TYPE if_BitCommand_u :
UNION
    awPBOM : ARRAY[0..1] OF WORD;
    dwPBOM : DWORD;
END_UNION
END_TYPE

(* stored: Version 1.1.0.1, ProductVersion 3.1.4024.6
   DUT if_BitCommand_u: Id {f6835c1c-7810-44c6-84a1-28d63c3de89e} *)
